FUNCTION_BLOCK OutputParameter
VAR_INPUT
  new_position, new_velocity, new_acceleration : ARRAY[0..ParameterList.maximumDegreeOfFreedom] OF LREAL;
  new_calculation : BOOL;
  calculation_duration : REAL; // us
  trajectory : Trajectory;
  current_time : LREAL;
  has_changed : BOOL;
END_VAR

END_FUNCTION_BLOCK

(* stored: Version 1.1.0.1, ProductVersion 3.1.4024.6
   POU OutputParameter: Id {597621a9-5523-4c13-96bf-7b02710f89f6}, SpecialFunc None *)
